// SIMATIC S7-200 SMART project (STEP 7-Micro/WIN SMART), CPU SR40

SYMBOL_TABLE 系统符号
Always_On        SM0.0    // 始终接通
END_SYMBOL_TABLE

ORGANIZATION_BLOCK MAIN:OB1
TITLE=程序注释
BEGIN
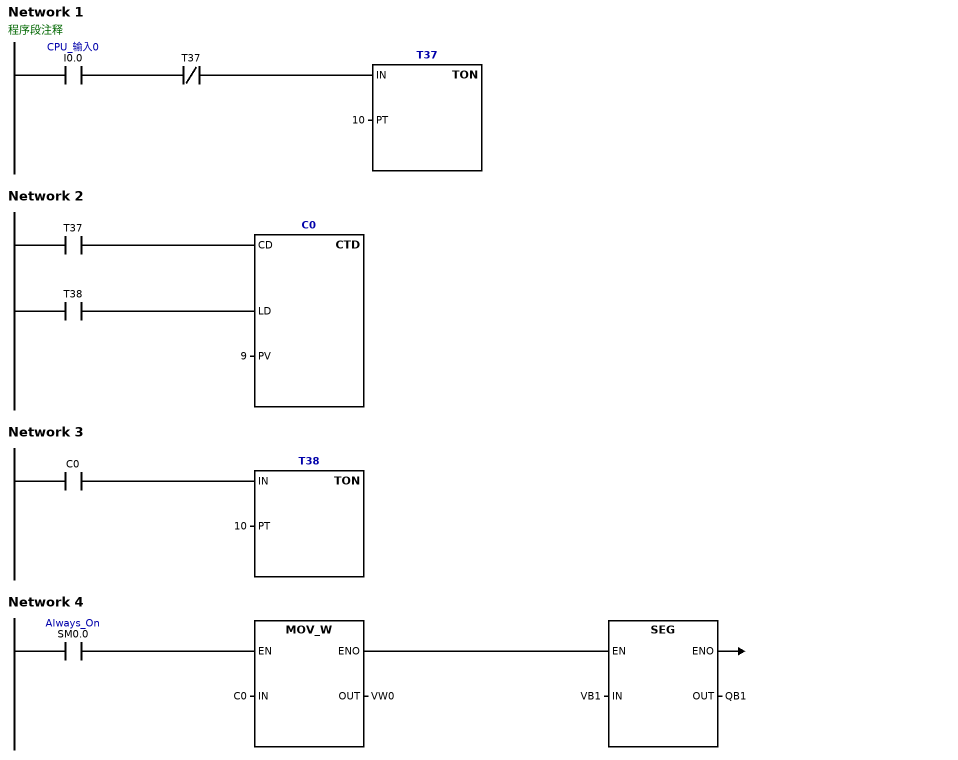
Network 1
// 程序段注释
LD     CPU_输入0:I0.0
AN     T37
TON    T37, 10
Network 2
LD     T37
LD     T38
CTD    C0, 9
Network 3
LD     C0
TON    T38, 10
Network 4
LD     Always_On:SM0.0
MOVW   C0, VW0
AENO
SEG    VB1, QB1
END_ORGANIZATION_BLOCK
